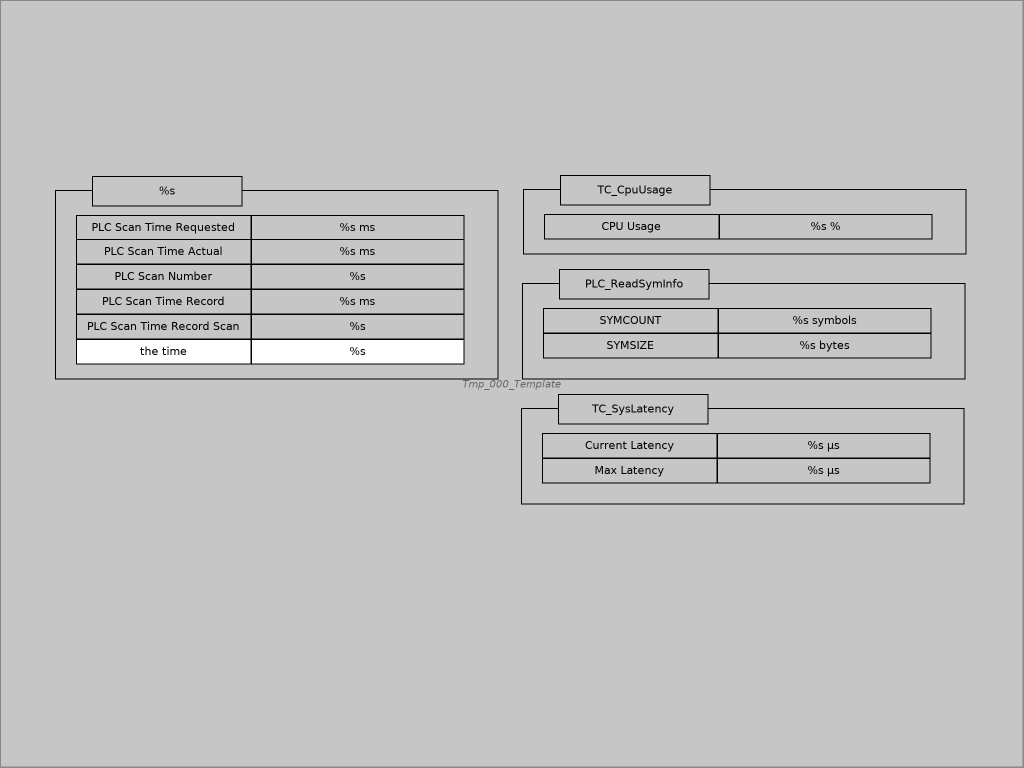
VISUALIZATION Sys_901_HMISystem  // 1024x768
    Frame (0,0 1024x768)
        shows Tmp_000_Template(header := gHMIData.hmiHeader)
    Rectangle (251,215 213x25), "%s ms", text variable: System.ScanTimeReq, text list: ''
    Rectangle (76,215 175x25), "PLC Scan Time Requested"
    Rectangle (76,239 175x25), "PLC Scan Time Actual"
    Rectangle (251,239 213x25), "%s ms", text variable: System.ScanTimeAct, text list: ''
    Rectangle (76,264 175x25), "PLC Scan Number"
    Rectangle (251,264 213x25), "%s", text variable: System.myPlcInfoTask1.CycleCount, text list: ''
    Rectangle (55,190 443x189)
    Rectangle (92,176 150x30), "%s", text variable: System.myPlcInfoTask1.TaskName
    Rectangle (76,289 175x25), "PLC Scan Time Record"
    Rectangle (251,289 213x25), "%s ms", text variable: System.ScanTimeRecord, text list: ''
    Rectangle (76,314 175x25), "PLC Scan Time Record Scan"
    Rectangle (251,314 213x25), "%s", text variable: System.ScanTimeRecordScan, text list: ''
    Rectangle (251,339 213x25), "%s", text variable: System.timeDT
    Rectangle (76,339 175x25), "the time"
    Rectangle (719,214 213x25), "%s %", text variable: System.cpuusageval, text list: ''
    Rectangle (544,214 175x25), "CPU Usage"
    Rectangle (523,189 443x65)
    Rectangle (560,175 150x30), "TC_CpuUsage"
    Rectangle (718,308 213x25), "%s symbols", text variable: System.symCount, text list: ''
    Rectangle (543,308 175x25), "SYMCOUNT"
    Rectangle (522,283 443x96)
    Rectangle (559,269 150x30), "PLC_ReadSymInfo"
    Rectangle (718,333 213x25), "%s bytes", text variable: System.sysSize, text list: ''
    Rectangle (543,333 175x25), "SYMSIZE"
    Rectangle (717,433 213x25), "%s µs", text variable: System.LatencyMicroSec, text list: ''
    Rectangle (542,433 175x25), "Current Latency"
    Rectangle (521,408 443x96)
    Rectangle (558,394 150x30), "TC_SysLatency"
    Rectangle (717,458 213x25), "%s µs", text variable: System.MaxLatencyMicroSec, text list: ''
    Rectangle (542,458 175x25), "Max Latency"
END_VISUALIZATION

(* stored: Version 1.1.0.1, ProductVersion 3.1.4024.12
   Visu Sys_901_HMISystem: Id {785d049b-80ed-4444-aba2-927731f3e4a5} *)
